// TIA Portal V18 export
TYPE "MEStoPLC_RecipeData_OP220"
// stored: IsFailsafeCompliant false
   STRUCT
      "M-PartType" : String[28];   // MES反馈产品型号，与PC测试交互使用
      "M-PartTypeRecordNr" : Int;   // 备选方案2：MES反馈配方记录号，采用数据记录号的方式，与PC测试交互使用
      "M-RecipeVer" : String[18];   // 工艺参数版本号
      "M-RecipeParameter" : "MEStoPLC_RecipeParameter_OP220";   // 工艺参数-判定阀值或设定目标值，配方是包含版本号和程序号的
      Reserve : Array[1..1436] of Byte;   // 配方数据预留
   END_STRUCT;
END_TYPE
